// TIA Portal project "Multistage Conveyor" (V17)
// Multistage Conveyor
// When a start button is ON, then
// The first Stage Motor runs for 10 seconds, then stops. After a 5 seconds delay, the second stage motor runs for 20 seconds and then the third stage motor will run for 15 seconds.

(* hardware
DEVICE "S7-1200 station_1"  S7-1200 Station
   slot 0: "Rack_0"  S7-1200 Rack  Rack  V1.0
   slot 1: "PLC_1"  CPU 1217C DC/DC/DC  6ES7 217-1AG40-0XB0  V4.5
*)

// ===== PLC "PLC_1"  CPU 1217C DC/DC/DC =====

VAR_GLOBAL   // PLC tag table "Default tag table"
   "Start_PB" AT %I0.1 : Bool;
   "M1" AT %Q0.0 : Bool;
   "M2" AT %Q0.1 : Bool;
   "M3" AT %Q0.2 : Bool;
   "Stop" AT %I0.0 : Bool;
   "Tag_1" AT %M0.0 : Bool;
   "Tag_2" AT %M0.2 : Bool;
   "Tag_3" AT %M0.3 : Bool;
END_VAR

// folder: System blocks/Program resources

DATA_BLOCK "IEC_Timer_0_DB"   // DB1
{ S7_Optimized_Access := 'TRUE' }
AUTHOR : Simatic
FAMILY : IEC
NAME : IEC_TMR
VERSION : 1.0
// stored: InstanceOfName IEC_TIMER
"IEC_TIMER"
BEGIN
END_DATA_BLOCK

DATA_BLOCK "IEC_Timer_0_DB_1"   // DB2
{ S7_Optimized_Access := 'TRUE' }
AUTHOR : Simatic
FAMILY : IEC
NAME : IEC_TMR
VERSION : 1.0
// stored: InstanceOfName IEC_TIMER
"IEC_TIMER"
BEGIN
END_DATA_BLOCK

DATA_BLOCK "IEC_Timer_0_DB_2"   // DB3
{ S7_Optimized_Access := 'TRUE' }
AUTHOR : Simatic
FAMILY : IEC
NAME : IEC_TMR
VERSION : 1.0
// stored: InstanceOfName IEC_TIMER
"IEC_TIMER"
BEGIN
END_DATA_BLOCK

DATA_BLOCK "IEC_Timer_0_DB_3"   // DB4
{ S7_Optimized_Access := 'TRUE' }
AUTHOR : Simatic
FAMILY : IEC
NAME : IEC_TMR
VERSION : 1.0
// stored: InstanceOfName IEC_TIMER
"IEC_TIMER"
BEGIN
END_DATA_BLOCK

DATA_BLOCK "IEC_Timer_0_DB_4"   // DB5
{ S7_Optimized_Access := 'TRUE' }
AUTHOR : Simatic
FAMILY : IEC
NAME : IEC_TMR
VERSION : 1.0
// stored: InstanceOfName IEC_TIMER
"IEC_TIMER"
BEGIN
END_DATA_BLOCK

DATA_BLOCK "IEC_Timer_0_DB_5"   // DB6
{ S7_Optimized_Access := 'TRUE' }
AUTHOR : Simatic
FAMILY : IEC
NAME : IEC_TMR
VERSION : 1.0
// stored: InstanceOfName IEC_TIMER
"IEC_TIMER"
BEGIN
END_DATA_BLOCK

DATA_BLOCK "IEC_Timer_0_DB_6"   // DB7
{ S7_Optimized_Access := 'TRUE' }
AUTHOR : Simatic
FAMILY : IEC
NAME : IEC_TMR
VERSION : 1.0
// stored: InstanceOfName IEC_TIMER
"IEC_TIMER"
BEGIN
END_DATA_BLOCK

// folder: (top level)

ORGANIZATION_BLOCK "Main"   // OB1, LAD, ProgramCycle
TITLE = "Main Program Sweep (Cycle)"
{ S7_Optimized_Access := 'TRUE' }
VERSION : 0.1
   VAR_INPUT
      Initial_Call : Bool;   // Initial call of this OB
      Remanence : Bool;   // =True, if remanent data are available
   END_VAR
BEGIN

REGION Network 1
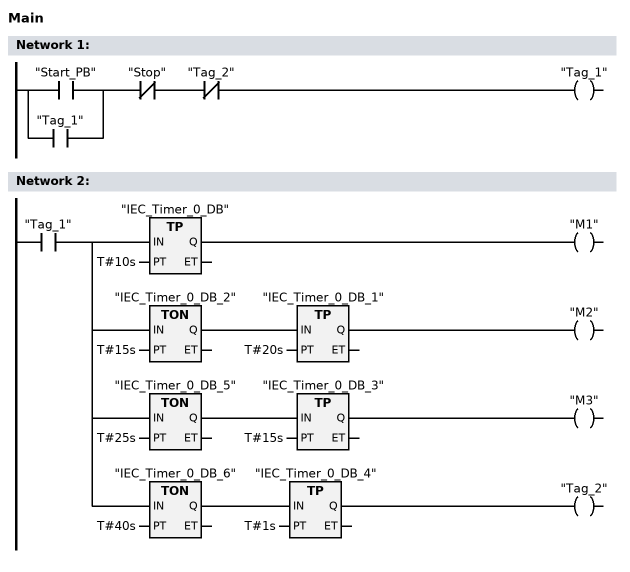
   RUNG wire#powerrail
      Contact( "Start_PB" )
      wire#w1
      I_Contact( "Stop" )
      I_Contact( "Tag_2" )
      Coil( "Tag_1" )
   END_RUNG
   RUNG wire#powerrail
      Contact( "Tag_1" )
   END_RUNG wire#w1
   // the same network as SCL:
   "Tag_1" := ("Start_PB" OR "Tag_1") AND NOT "Stop" AND NOT "Tag_2";
END_REGION

REGION Network 2
   "IEC_Timer_0_DB".TP(IN := "Tag_1", PT := T#10s);
   "M1" := "IEC_Timer_0_DB".Q;
   "IEC_Timer_0_DB_2".TON(IN := "Tag_1", PT := T#15s);
   "IEC_Timer_0_DB_1".TP(IN := "IEC_Timer_0_DB_2".Q, PT := T#20s);
   "M2" := "IEC_Timer_0_DB_1".Q;
   "IEC_Timer_0_DB_5".TON(IN := "Tag_1", PT := T#25s);
   "IEC_Timer_0_DB_3".TP(IN := "IEC_Timer_0_DB_5".Q, PT := T#15s);
   "M3" := "IEC_Timer_0_DB_3".Q;
   "IEC_Timer_0_DB_6".TON(IN := "Tag_1", PT := T#40s);
   "IEC_Timer_0_DB_4".TP(IN := "IEC_Timer_0_DB_6".Q, PT := T#1s);
   "Tag_2" := "IEC_Timer_0_DB_4".Q;
END_REGION
END_ORGANIZATION_BLOCK